// TwinCAT 3 PLC project PLC
// ProgramVersion: 3.1.4024.0
// libraries:
//   Tc2_MC2, * (Beckhoff Automation GmbH)
//   Tc2_Standard, * (Beckhoff Automation GmbH)
//   Tc2_System, * (Beckhoff Automation GmbH)
//   Tc3_Module, * (Beckhoff Automation GmbH)
// project tree:
//   DUTs/ E_States.TcDUT
//   GVLs/ GVL.TcGVL
//   / PlcTask.TcTTO
//   POUs/ FB_StateMachine.TcPOU, MAIN.TcPOU
// real-time tasks:
//   TASK PlcTask: cycle T#10ms, priority 20, ADS port 350
//   TASK PlcTask1: cycle T#10ms, priority 21, ADS port 351
// motion (NC):
//   TASK NC-Task 1 SAF: cycle T#2ms, priority 4, ADS port 501
//   TASK NC-Task 1 SVB: cycle T#10ms, priority 8, ADS port 511
//   AXIS Asse 1 (id 1)
//     OtherSettings: AllowMotionCmdToSlave=true
//     encoder EncType=1
//     drive DrvType=5
//       Analog: TorqueSetpointScale=10, ScaleFactorActTorque=0.1
//     controller CtrType=1
//       CtrPara: PriorControlFactor=1
//         Observer: BandWidth=20
// variable links:
//   PLC/PLC Instance <-> NC-Task 1 SAF/Axes/Asse 1
//     PlcTask Inputs/GVL.axis.NcToPlc <-> Outputs/ToPlc
//     PlcTask Outputs/GVL.axis.PlcToNc <-> Inputs/FromPlc

CONFIGURATION PLC
    RESOURCE PLC ON TwinCAT3
        TASK PlcTask(INTERVAL := T#10ms, PRIORITY := 21);
        PROGRAM MAIN WITH PlcTask : MAIN;
    END_RESOURCE
END_CONFIGURATION

// ---- DUTs/E_States.TcDUT
{attribute 'qualified_only'}
{attribute 'strict'}
TYPE E_States :
(
	eClosed := 0,
	eOpened,
	eOpening,
	eClosing
);
END_TYPE

// ---- GVLs/GVL.TcGVL
{attribute 'qualified_only'}
VAR_GLOBAL
	//Input
	bUltrasonicSensor: BOOL;
	bUpperLimitSwitch: BOOL;
	bLowerLimitSwitch: BOOL;
	bPhotocell: BOOL;
	//Output
	nMotorPosition: LREAL;
	bMotorUp: BOOL;
	bMotorDown: BOOL;
	//Internal
	axis: AXIS_REF;
	fBJog: MC_Jog;
	fBPower: MC_Power;
END_VAR

// ---- POUs/MAIN.TcPOU
PROGRAM MAIN
VAR
	StateMachine: FB_StateMachine;
END_VAR

//Invoco macchina a stati
StateMachine(bUltrasonicSensor:= GVL.bUltrasonicSensor, bUpperLimitSwitch:= GVL.bUpperLimitSwitch, bLowerLimitSwitch:= GVL.bLowerLimitSwitch, bPhotocell:= GVL.bPhotocell );
//Scrittura variabili Output
GVL.bMotorUp := StateMachine.bMotorUp;
GVL.bMotorDown := StateMachine.bMotorDown;
GVL.nMotorPosition := GVL.axis.NcToPlc.ActPos;
//Movimentazione motore
GVL.fBPower(Axis:=GVL.axis, Enable:=TRUE, Enable_Positive:= GVL.bMotorUp, Enable_Negative:= GVL.bMotorDown, Override:=100);
GVL.fBJog(Axis:=GVL.axis, JogForward:= GVL.bMotorUp, JogBackwards:= GVL.bMotorDown, Velocity:=100);

END_PROGRAM

// ---- POUs/FB_StateMachine.TcPOU
FUNCTION_BLOCK FB_StateMachine
VAR_INPUT
	bUltrasonicSensor: BOOL;
	bUpperLimitSwitch: BOOL;
	bLowerLimitSwitch: BOOL;
	bPhotocell: BOOL;
END_VAR
VAR_OUTPUT
	bMotorUp: BOOL;
	bMotorDown: BOOL;
END_VAR
VAR
	bTimeExpired: BOOL;
	fBTon: TON;
	state : E_States;
END_VAR

CASE state OF
	E_States.eClosed:
		bMotorUp := FALSE;
		bMotorDown := FALSE;
		IF bUltrasonicSensor THEN
			state:= E_States.eOpening;
		END_IF
	
	E_States.eOpening:
		bMotorUp := TRUE;
		bMotorDown := FALSE;
		IF bUpperLimitSwitch THEN
			state:= E_States.eOpened;
		END_IF

	E_States.eOpened:
		fBTon(IN := NOT bPhotocell AND NOT bUltrasonicSensor , PT:=T#5S , Q=>, ET=> );
		bMotorUp := FALSE;
		bMotorDown := FALSE;
		IF fBTon.Q THEN
			state:= E_States.eClosing;
		END_IF
	
	E_States.eClosing:
		fBTon(IN := FALSE);
		bMotorUp := FALSE;
		bMotorDown := TRUE;
		IF bPhotocell OR bUltrasonicSensor THEN
			state:= E_States.eOpening;
		ELSIF bLowerLimitSwitch THEN
			state:= E_States.eClosed;
		END_IF
END_CASE

END_FUNCTION_BLOCK
